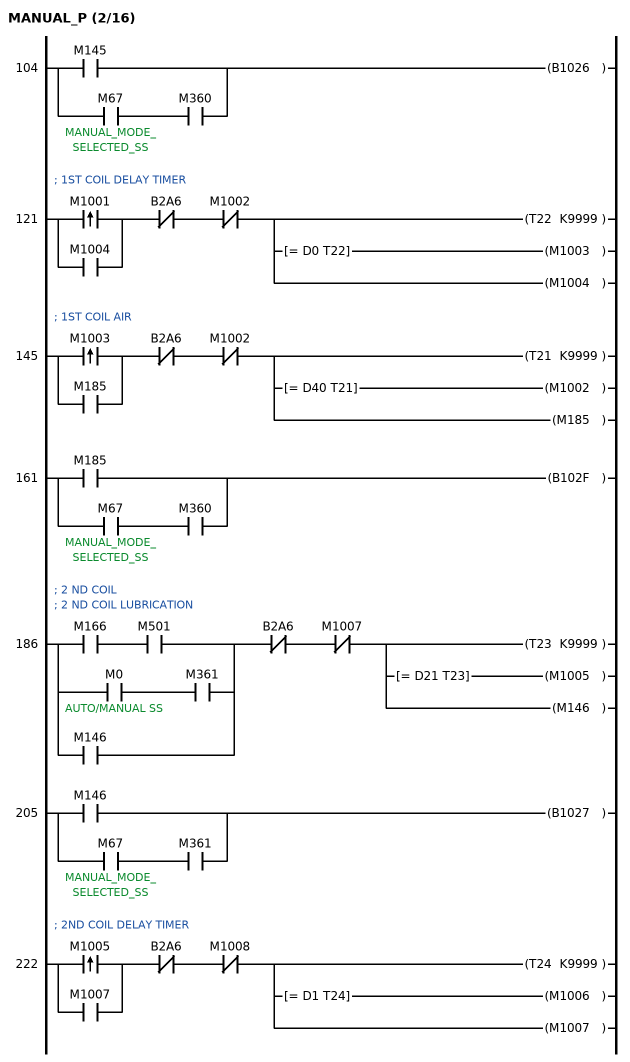
[picture p24: ladder of MANUAL_P, rungs at steps 104 to 222]
104   LD      M145
      LD      M67  ; MANUAL_MODE_SELECTED_SS
      AND     M360
      ORB
      OUT     B1026
; 1ST COIL DELAY TIMER
121   LDP     M1001
      OR      M1004
      ANI     B2A6
      ANI     M1002
      OUT     T22 K9999
      MPS
      AND=    D0 T22
      OUT     M1003
      MPP
      OUT     M1004
; 1ST COIL AIR
145   LDP     M1003
      OR      M185
      ANI     B2A6
      ANI     M1002
      OUT     T21 K9999
      MPS
      AND=    D40 T21
      OUT     M1002
      MPP
      OUT     M185
161   LD      M185
      LD      M67  ; MANUAL_MODE_SELECTED_SS
      AND     M360
      ORB
      OUT     B102F
; 2 ND COIL
; 2 ND COIL LUBRICATION
186   LD      M166
      AND     M501
      LD      M0  ; AUTO/MANUAL SS
      AND     M361
      ORB
      OR      M146
      ANI     B2A6
      ANI     M1007
      OUT     T23 K9999
      MPS
      AND=    D21 T23
      OUT     M1005
      MPP
      OUT     M146
205   LD      M146
      LD      M67  ; MANUAL_MODE_SELECTED_SS
      AND     M361
      ORB
      OUT     B1027
; 2ND COIL DELAY TIMER
222   LDP     M1005
      OR      M1007
      ANI     B2A6
      ANI     M1008
      OUT     T24 K9999
      MPS
      AND=    D1 T24
      OUT     M1006
      MPP
      OUT     M1007
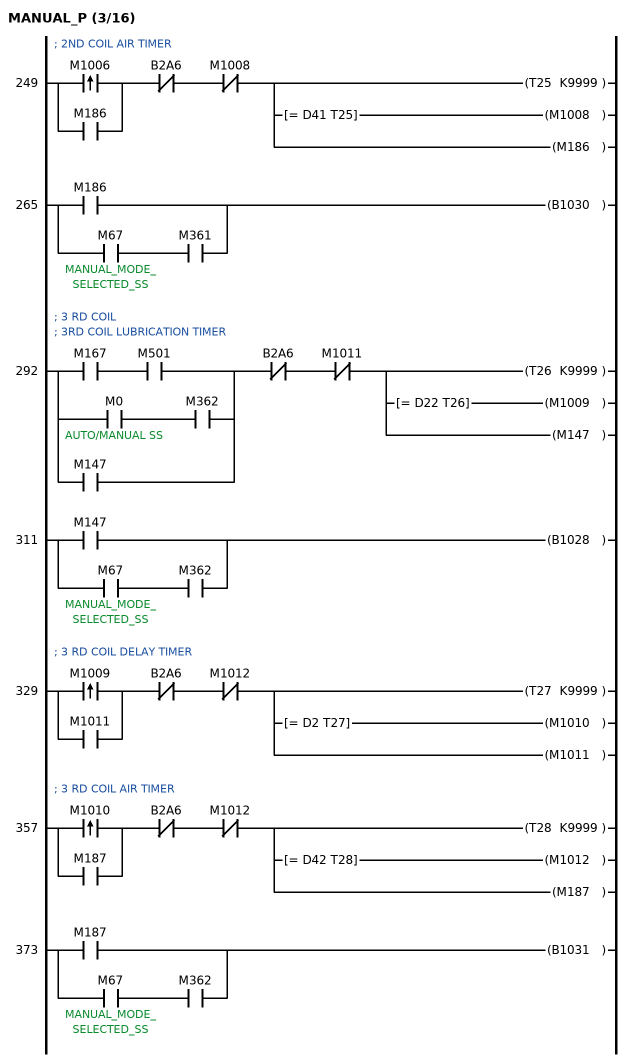
; 2ND COIL AIR TIMER
249   LDP     M1006
      OR      M186
      ANI     B2A6
      ANI     M1008
      OUT     T25 K9999
      MPS
      AND=    D41 T25
      OUT     M1008
      MPP
      OUT     M186
265   LD      M186
      LD      M67  ; MANUAL_MODE_SELECTED_SS
      AND     M361
      ORB
      OUT     B1030
; 3 RD COIL
; 3RD COIL LUBRICATION TIMER
292   LD      M167
      AND     M501
      LD      M0  ; AUTO/MANUAL SS
      AND     M362
      ORB
      OR      M147
      ANI     B2A6
      ANI     M1011
      OUT     T26 K9999
      MPS
      AND=    D22 T26
      OUT     M1009
      MPP
      OUT     M147
311   LD      M147
      LD      M67  ; MANUAL_MODE_SELECTED_SS
      AND     M362
      ORB
      OUT     B1028
; 3 RD COIL DELAY TIMER
329   LDP     M1009
      OR      M1011
      ANI     B2A6
      ANI     M1012
      OUT     T27 K9999
      MPS
      AND=    D2 T27
      OUT     M1010
      MPP
      OUT     M1011
; 3 RD COIL AIR TIMER
357   LDP     M1010
      OR      M187
      ANI     B2A6
      ANI     M1012
      OUT     T28 K9999
      MPS
      AND=    D42 T28
      OUT     M1012
      MPP
      OUT     M187
373   LD      M187
      LD      M67  ; MANUAL_MODE_SELECTED_SS
      AND     M362
      ORB
      OUT     B1031
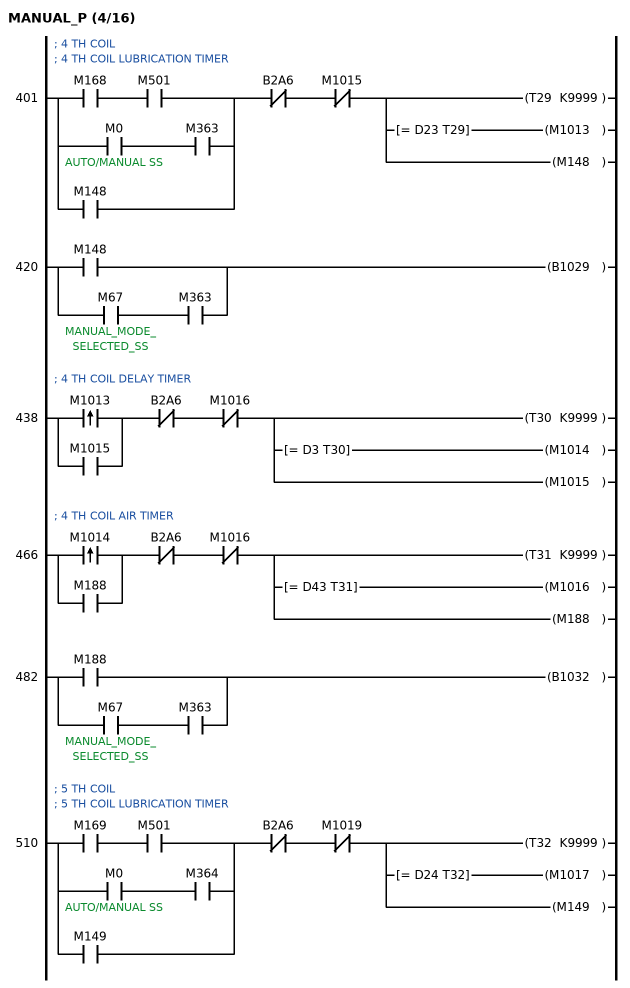
; 4 TH COIL
; 4 TH COIL LUBRICATION TIMER
401   LD      M168
      AND     M501
      LD      M0  ; AUTO/MANUAL SS
      AND     M363
      ORB
      OR      M148
      ANI     B2A6
      ANI     M1015
      OUT     T29 K9999
      MPS
      AND=    D23 T29
      OUT     M1013
      MPP
      OUT     M148
420   LD      M148
      LD      M67  ; MANUAL_MODE_SELECTED_SS
      AND     M363
      ORB
      OUT     B1029
; 4 TH COIL DELAY TIMER
438   LDP     M1013
      OR      M1015
      ANI     B2A6
      ANI     M1016
      OUT     T30 K9999
      MPS
      AND=    D3 T30
      OUT     M1014
      MPP
      OUT     M1015
; 4 TH COIL AIR TIMER
466   LDP     M1014
      OR      M188
      ANI     B2A6
      ANI     M1016
      OUT     T31 K9999
      MPS
      AND=    D43 T31
      OUT     M1016
      MPP
      OUT     M188
482   LD      M188
      LD      M67  ; MANUAL_MODE_SELECTED_SS
      AND     M363
      ORB
      OUT     B1032
; 5 TH COIL
; 5 TH COIL LUBRICATION TIMER
510   LD      M169
      AND     M501
      LD      M0  ; AUTO/MANUAL SS
      AND     M364
      ORB
      OR      M149
      ANI     B2A6
      ANI     M1019
      OUT     T32 K9999
      MPS
      AND=    D24 T32
      OUT     M1017
      MPP
      OUT     M149
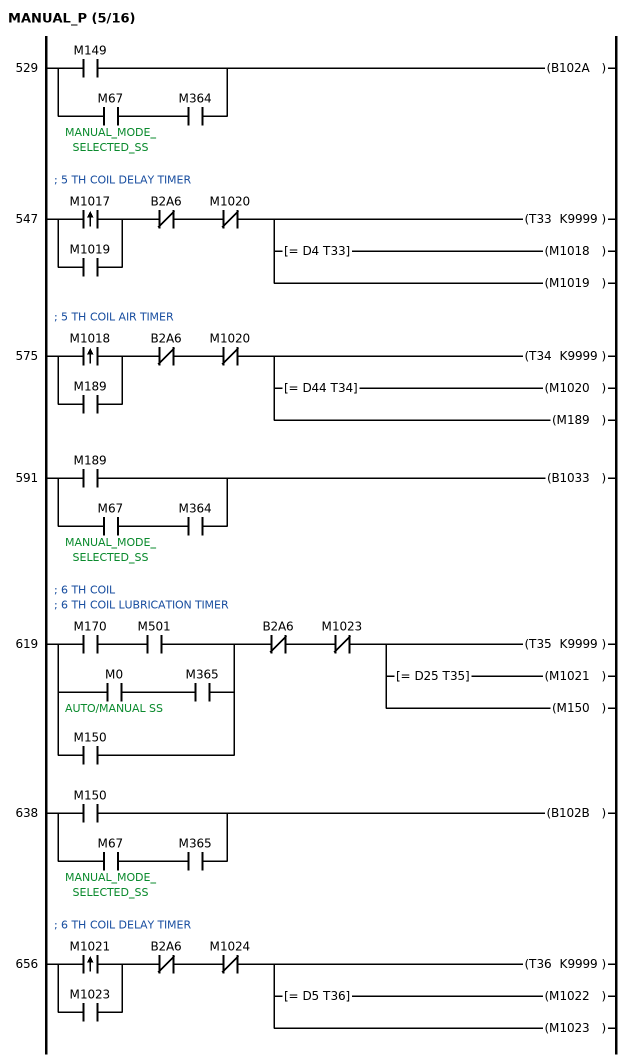
529   LD      M149
      LD      M67  ; MANUAL_MODE_SELECTED_SS
      AND     M364
      ORB
      OUT     B102A
; 5 TH COIL DELAY TIMER
547   LDP     M1017
      OR      M1019
      ANI     B2A6
      ANI     M1020
      OUT     T33 K9999
      MPS
      AND=    D4 T33
      OUT     M1018
      MPP
      OUT     M1019
; 5 TH COIL AIR TIMER
575   LDP     M1018
      OR      M189
      ANI     B2A6
      ANI     M1020
      OUT     T34 K9999
      MPS
      AND=    D44 T34
      OUT     M1020
      MPP
      OUT     M189
591   LD      M189
      LD      M67  ; MANUAL_MODE_SELECTED_SS
      AND     M364
      ORB
      OUT     B1033
; 6 TH COIL
; 6 TH COIL LUBRICATION TIMER
619   LD      M170
      AND     M501
      LD      M0  ; AUTO/MANUAL SS
      AND     M365
      ORB
      OR      M150
      ANI     B2A6
      ANI     M1023
      OUT     T35 K9999
      MPS
      AND=    D25 T35
      OUT     M1021
      MPP
      OUT     M150
638   LD      M150
      LD      M67  ; MANUAL_MODE_SELECTED_SS
      AND     M365
      ORB
      OUT     B102B
; 6 TH COIL DELAY TIMER
656   LDP     M1021
      OR      M1023
      ANI     B2A6
      ANI     M1024
      OUT     T36 K9999
      MPS
      AND=    D5 T36
      OUT     M1022
      MPP
      OUT     M1023
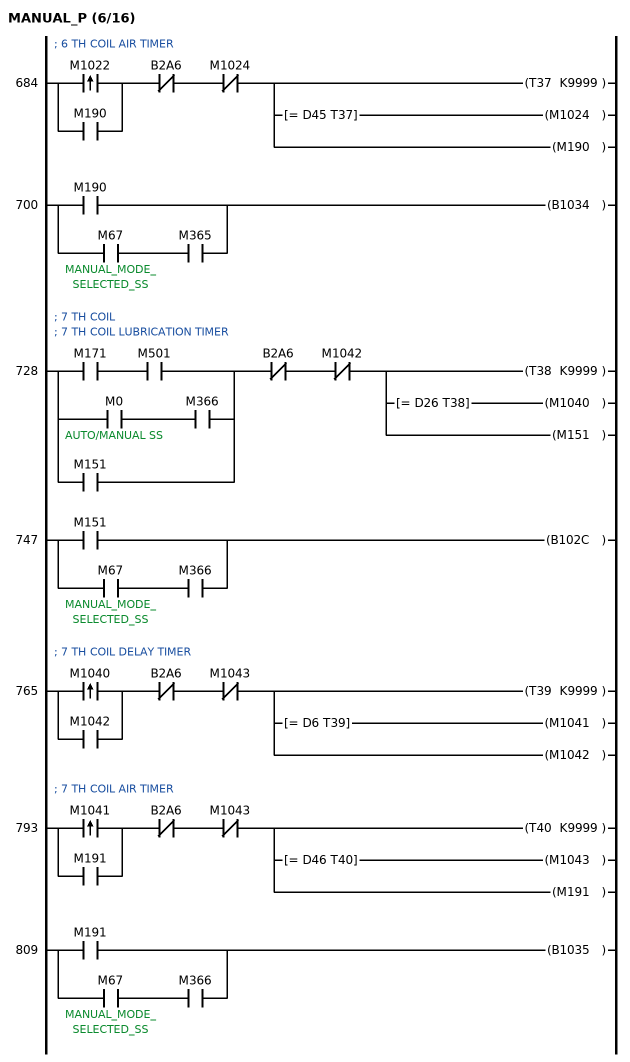
; 6 TH COIL AIR TIMER
684   LDP     M1022
      OR      M190
      ANI     B2A6
      ANI     M1024
      OUT     T37 K9999
      MPS
      AND=    D45 T37
      OUT     M1024
      MPP
      OUT     M190
700   LD      M190
      LD      M67  ; MANUAL_MODE_SELECTED_SS
      AND     M365
      ORB
      OUT     B1034
; 7 TH COIL
; 7 TH COIL LUBRICATION TIMER
728   LD      M171
      AND     M501
      LD      M0  ; AUTO/MANUAL SS
      AND     M366
      ORB
      OR      M151
      ANI     B2A6
      ANI     M1042
      OUT     T38 K9999
      MPS
      AND=    D26 T38
      OUT     M1040
      MPP
      OUT     M151
747   LD      M151
      LD      M67  ; MANUAL_MODE_SELECTED_SS
      AND     M366
      ORB
      OUT     B102C
; 7 TH COIL DELAY TIMER
765   LDP     M1040
      OR      M1042
      ANI     B2A6
      ANI     M1043
      OUT     T39 K9999
      MPS
      AND=    D6 T39
      OUT     M1041
      MPP
      OUT     M1042
; 7 TH COIL AIR TIMER
793   LDP     M1041
      OR      M191
      ANI     B2A6
      ANI     M1043
      OUT     T40 K9999
      MPS
      AND=    D46 T40
      OUT     M1043
      MPP
      OUT     M191
809   LD      M191
      LD      M67  ; MANUAL_MODE_SELECTED_SS
      AND     M366
      ORB
      OUT     B1035
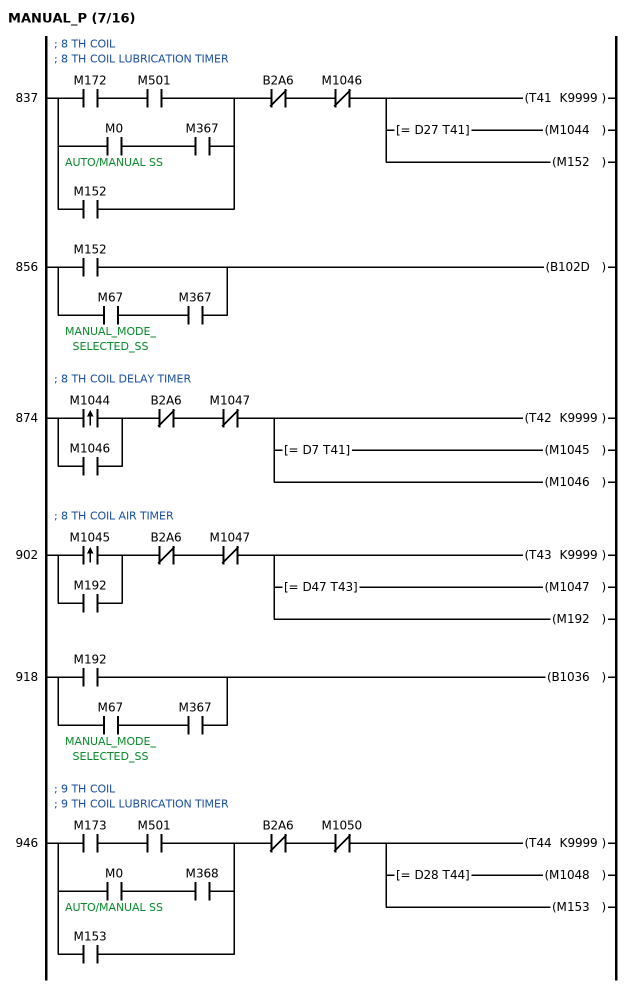
; 8 TH COIL
; 8 TH COIL LUBRICATION TIMER
837   LD      M172
      AND     M501
      LD      M0  ; AUTO/MANUAL SS
      AND     M367
      ORB
      OR      M152
      ANI     B2A6
      ANI     M1046
      OUT     T41 K9999
      MPS
      AND=    D27 T41
      OUT     M1044
      MPP
      OUT     M152
856   LD      M152
      LD      M67  ; MANUAL_MODE_SELECTED_SS
      AND     M367
      ORB
      OUT     B102D
; 8 TH COIL DELAY TIMER
874   LDP     M1044
      OR      M1046
      ANI     B2A6
      ANI     M1047
      OUT     T42 K9999
      MPS
      AND=    D7 T41
      OUT     M1045
      MPP
      OUT     M1046
; 8 TH COIL AIR TIMER
902   LDP     M1045
      OR      M192
      ANI     B2A6
      ANI     M1047
      OUT     T43 K9999
      MPS
      AND=    D47 T43
      OUT     M1047
      MPP
      OUT     M192
918   LD      M192
      LD      M67  ; MANUAL_MODE_SELECTED_SS
      AND     M367
      ORB
      OUT     B1036
; 9 TH COIL
; 9 TH COIL LUBRICATION TIMER
946   LD      M173
      AND     M501
      LD      M0  ; AUTO/MANUAL SS
      AND     M368
      ORB
      OR      M153
      ANI     B2A6
      ANI     M1050
      OUT     T44 K9999
      MPS
      AND=    D28 T44
      OUT     M1048
      MPP
      OUT     M153
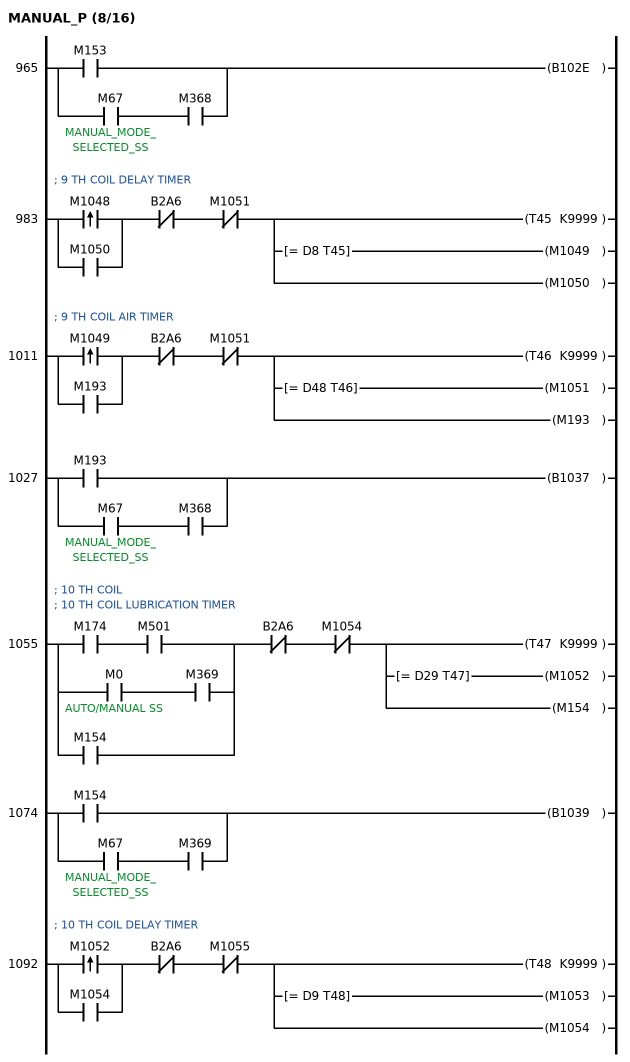
965   LD      M153
      LD      M67  ; MANUAL_MODE_SELECTED_SS
      AND     M368
      ORB
      OUT     B102E
; 9 TH COIL DELAY TIMER
983   LDP     M1048
      OR      M1050
      ANI     B2A6
      ANI     M1051
      OUT     T45 K9999
      MPS
      AND=    D8 T45
      OUT     M1049
      MPP
      OUT     M1050
; 9 TH COIL AIR TIMER
1011  LDP     M1049
      OR      M193
      ANI     B2A6
      ANI     M1051
      OUT     T46 K9999
      MPS
      AND=    D48 T46
      OUT     M1051
      MPP
      OUT     M193
1027  LD      M193
      LD      M67  ; MANUAL_MODE_SELECTED_SS
      AND     M368
      ORB
      OUT     B1037
; 10 TH COIL
; 10 TH COIL LUBRICATION TIMER
1055  LD      M174
      AND     M501
      LD      M0  ; AUTO/MANUAL SS
      AND     M369
      ORB
      OR      M154
      ANI     B2A6
      ANI     M1054
      OUT     T47 K9999
      MPS
      AND=    D29 T47
      OUT     M1052
      MPP
      OUT     M154
1074  LD      M154
      LD      M67  ; MANUAL_MODE_SELECTED_SS
      AND     M369
      ORB
      OUT     B1039
; 10 TH COIL DELAY TIMER
1092  LDP     M1052
      OR      M1054
      ANI     B2A6
      ANI     M1055
      OUT     T48 K9999
      MPS
      AND=    D9 T48
      OUT     M1053
      MPP
      OUT     M1054
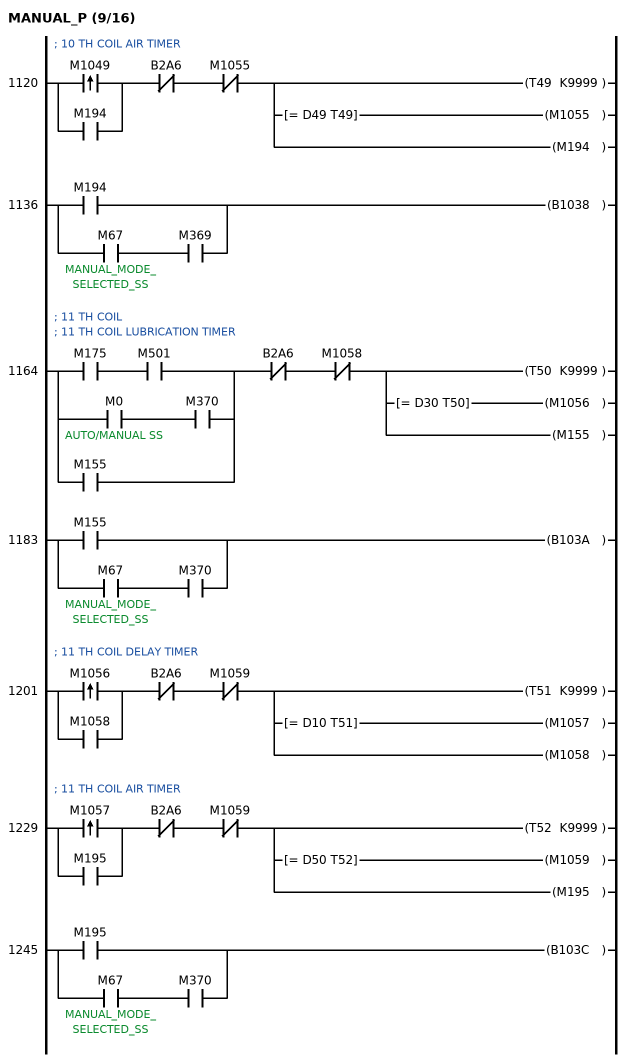
; 10 TH COIL AIR TIMER
1120  LDP     M1049
      OR      M194
      ANI     B2A6
      ANI     M1055
      OUT     T49 K9999
      MPS
      AND=    D49 T49
      OUT     M1055
      MPP
      OUT     M194
1136  LD      M194
      LD      M67  ; MANUAL_MODE_SELECTED_SS
      AND     M369
      ORB
      OUT     B1038
; 11 TH COIL
; 11 TH COIL LUBRICATION TIMER
1164  LD      M175
      AND     M501
      LD      M0  ; AUTO/MANUAL SS
      AND     M370
      ORB
      OR      M155
      ANI     B2A6
      ANI     M1058
      OUT     T50 K9999
      MPS
      AND=    D30 T50
      OUT     M1056
      MPP
      OUT     M155
1183  LD      M155
      LD      M67  ; MANUAL_MODE_SELECTED_SS
      AND     M370
      ORB
      OUT     B103A
; 11 TH COIL DELAY TIMER
1201  LDP     M1056
      OR      M1058
      ANI     B2A6
      ANI     M1059
      OUT     T51 K9999
      MPS
      AND=    D10 T51
      OUT     M1057
      MPP
      OUT     M1058
; 11 TH COIL AIR TIMER
1229  LDP     M1057
      OR      M195
      ANI     B2A6
      ANI     M1059
      OUT     T52 K9999
      MPS
      AND=    D50 T52
      OUT     M1059
      MPP
      OUT     M195
1245  LD      M195
      LD      M67  ; MANUAL_MODE_SELECTED_SS
      AND     M370
      ORB
      OUT     B103C
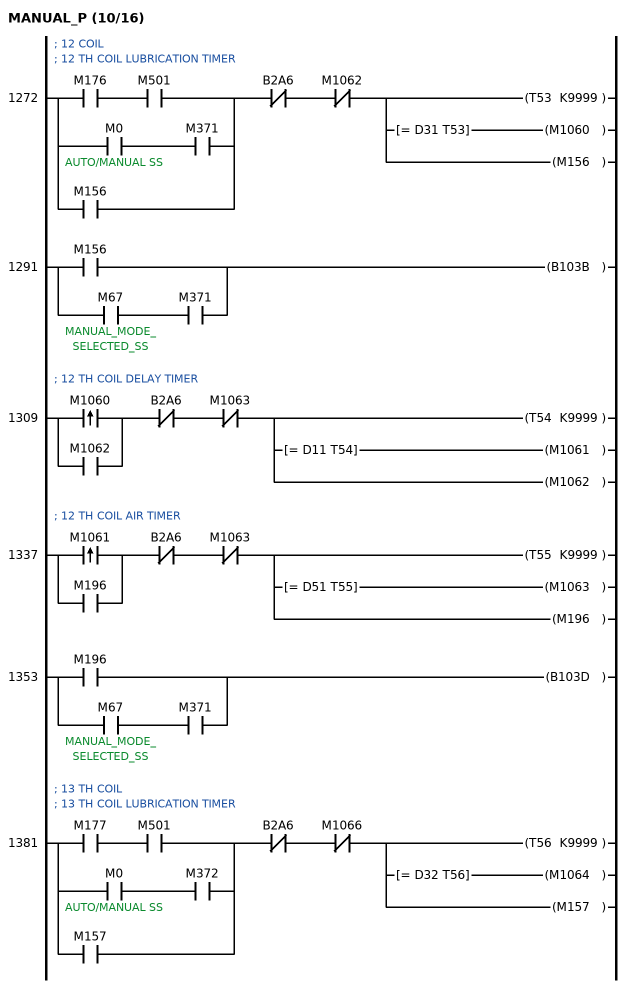
; 12 COIL
; 12 TH COIL LUBRICATION TIMER
1272  LD      M176
      AND     M501
      LD      M0  ; AUTO/MANUAL SS
      AND     M371
      ORB
      OR      M156
      ANI     B2A6
      ANI     M1062
      OUT     T53 K9999
      MPS
      AND=    D31 T53
      OUT     M1060
      MPP
      OUT     M156
1291  LD      M156
      LD      M67  ; MANUAL_MODE_SELECTED_SS
      AND     M371
      ORB
      OUT     B103B
; 12 TH COIL DELAY TIMER
1309  LDP     M1060
      OR      M1062
      ANI     B2A6
      ANI     M1063
      OUT     T54 K9999
      MPS
      AND=    D11 T54
      OUT     M1061
      MPP
      OUT     M1062
; 12 TH COIL AIR TIMER
1337  LDP     M1061
      OR      M196
      ANI     B2A6
      ANI     M1063
      OUT     T55 K9999
      MPS
      AND=    D51 T55
      OUT     M1063
      MPP
      OUT     M196
1353  LD      M196
      LD      M67  ; MANUAL_MODE_SELECTED_SS
      AND     M371
      ORB
      OUT     B103D
; 13 TH COIL
; 13 TH COIL LUBRICATION TIMER
1381  LD      M177
      AND     M501
      LD      M0  ; AUTO/MANUAL SS
      AND     M372
      ORB
      OR      M157
      ANI     B2A6
      ANI     M1066
      OUT     T56 K9999
      MPS
      AND=    D32 T56
      OUT     M1064
      MPP
      OUT     M157
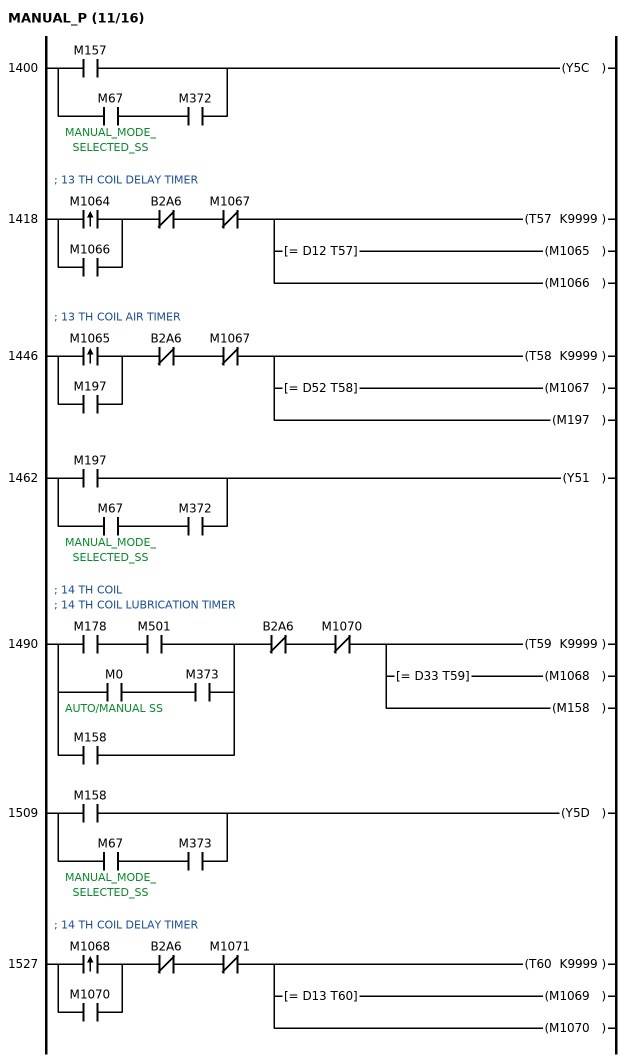
1400  LD      M157
      LD      M67  ; MANUAL_MODE_SELECTED_SS
      AND     M372
      ORB
      OUT     Y5C
; 13 TH COIL DELAY TIMER
1418  LDP     M1064
      OR      M1066
      ANI     B2A6
      ANI     M1067
      OUT     T57 K9999
      MPS
      AND=    D12 T57
      OUT     M1065
      MPP
      OUT     M1066
; 13 TH COIL AIR TIMER
1446  LDP     M1065
      OR      M197
      ANI     B2A6
      ANI     M1067
      OUT     T58 K9999
      MPS
      AND=    D52 T58
      OUT     M1067
      MPP
      OUT     M197
1462  LD      M197
      LD      M67  ; MANUAL_MODE_SELECTED_SS
      AND     M372
      ORB
      OUT     Y51
; 14 TH COIL
; 14 TH COIL LUBRICATION TIMER
1490  LD      M178
      AND     M501
      LD      M0  ; AUTO/MANUAL SS
      AND     M373
      ORB
      OR      M158
      ANI     B2A6
      ANI     M1070
      OUT     T59 K9999
      MPS
      AND=    D33 T59
      OUT     M1068
      MPP
      OUT     M158
1509  LD      M158
      LD      M67  ; MANUAL_MODE_SELECTED_SS
      AND     M373
      ORB
      OUT     Y5D
; 14 TH COIL DELAY TIMER
1527  LDP     M1068
      OR      M1070
      ANI     B2A6
      ANI     M1071
      OUT     T60 K9999
      MPS
      AND=    D13 T60
      OUT     M1069
      MPP
      OUT     M1070
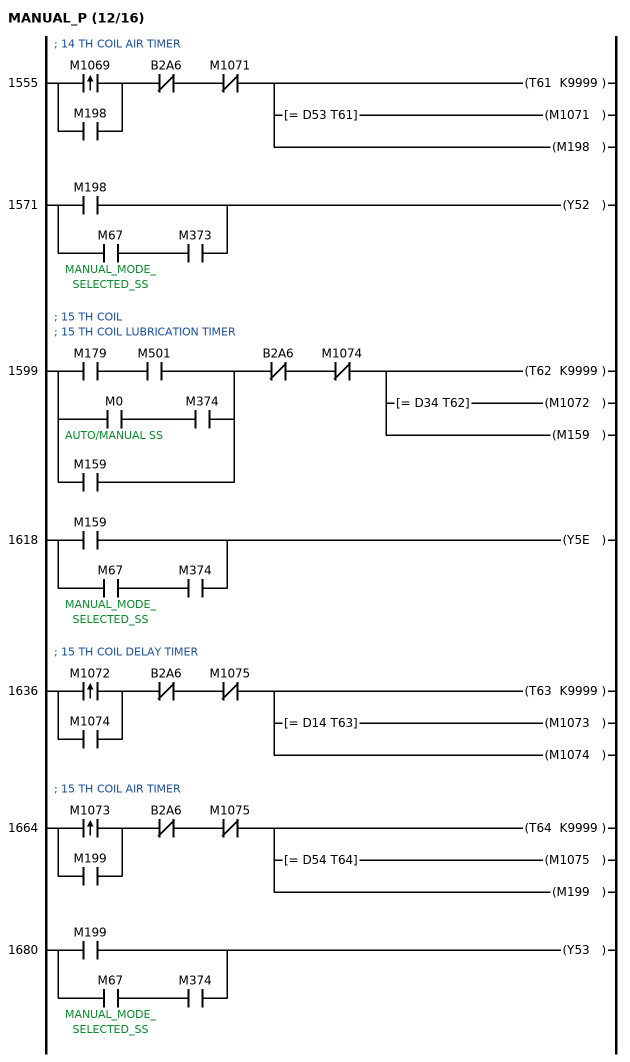
; 14 TH COIL AIR TIMER
1555  LDP     M1069
      OR      M198
      ANI     B2A6
      ANI     M1071
      OUT     T61 K9999
      MPS
      AND=    D53 T61
      OUT     M1071
      MPP
      OUT     M198
1571  LD      M198
      LD      M67  ; MANUAL_MODE_SELECTED_SS
      AND     M373
      ORB
      OUT     Y52
; 15 TH COIL
; 15 TH COIL LUBRICATION TIMER
1599  LD      M179
      AND     M501
      LD      M0  ; AUTO/MANUAL SS
      AND     M374
      ORB
      OR      M159
      ANI     B2A6
      ANI     M1074
      OUT     T62 K9999
      MPS
      AND=    D34 T62
      OUT     M1072
      MPP
      OUT     M159
1618  LD      M159
      LD      M67  ; MANUAL_MODE_SELECTED_SS
      AND     M374
      ORB
      OUT     Y5E
; 15 TH COIL DELAY TIMER
1636  LDP     M1072
      OR      M1074
      ANI     B2A6
      ANI     M1075
      OUT     T63 K9999
      MPS
      AND=    D14 T63
      OUT     M1073
      MPP
      OUT     M1074
; 15 TH COIL AIR TIMER
1664  LDP     M1073
      OR      M199
      ANI     B2A6
      ANI     M1075
      OUT     T64 K9999
      MPS
      AND=    D54 T64
      OUT     M1075
      MPP
      OUT     M199
1680  LD      M199
      LD      M67  ; MANUAL_MODE_SELECTED_SS
      AND     M374
      ORB
      OUT     Y53
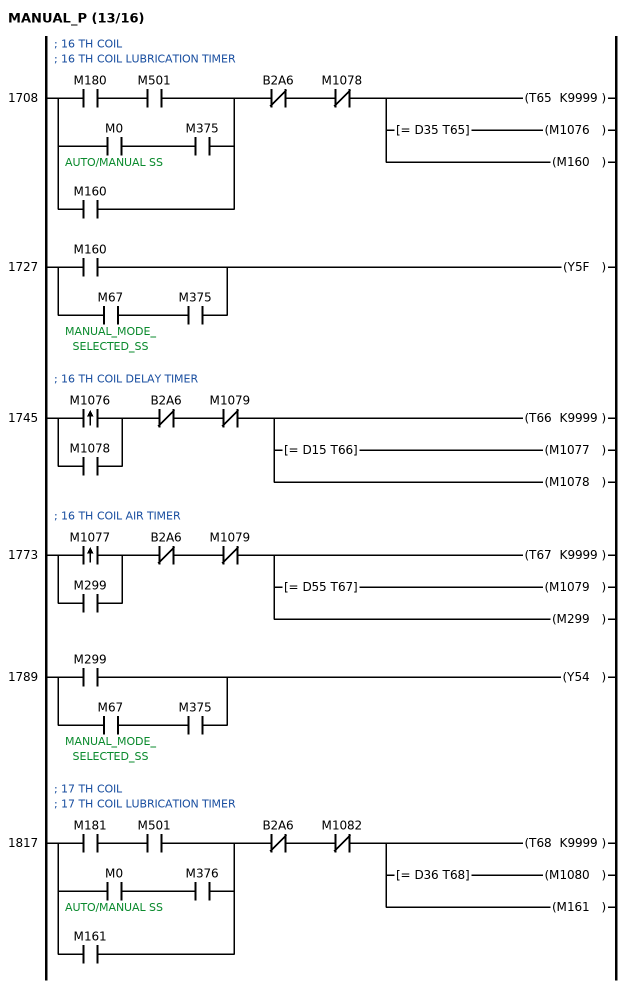
; 16 TH COIL
; 16 TH COIL LUBRICATION TIMER
1708  LD      M180
      AND     M501
      LD      M0  ; AUTO/MANUAL SS
      AND     M375
      ORB
      OR      M160
      ANI     B2A6
      ANI     M1078
      OUT     T65 K9999
      MPS
      AND=    D35 T65
      OUT     M1076
      MPP
      OUT     M160
1727  LD      M160
      LD      M67  ; MANUAL_MODE_SELECTED_SS
      AND     M375
      ORB
      OUT     Y5F
; 16 TH COIL DELAY TIMER
1745  LDP     M1076
      OR      M1078
      ANI     B2A6
      ANI     M1079
      OUT     T66 K9999
      MPS
      AND=    D15 T66
      OUT     M1077
      MPP
      OUT     M1078
; 16 TH COIL AIR TIMER
1773  LDP     M1077
      OR      M299
      ANI     B2A6
      ANI     M1079
      OUT     T67 K9999
      MPS
      AND=    D55 T67
      OUT     M1079
      MPP
      OUT     M299
1789  LD      M299
      LD      M67  ; MANUAL_MODE_SELECTED_SS
      AND     M375
      ORB
      OUT     Y54
; 17 TH COIL
; 17 TH COIL LUBRICATION TIMER
1817  LD      M181
      AND     M501
      LD      M0  ; AUTO/MANUAL SS
      AND     M376
      ORB
      OR      M161
      ANI     B2A6
      ANI     M1082
      OUT     T68 K9999
      MPS
      AND=    D36 T68
      OUT     M1080
      MPP
      OUT     M161
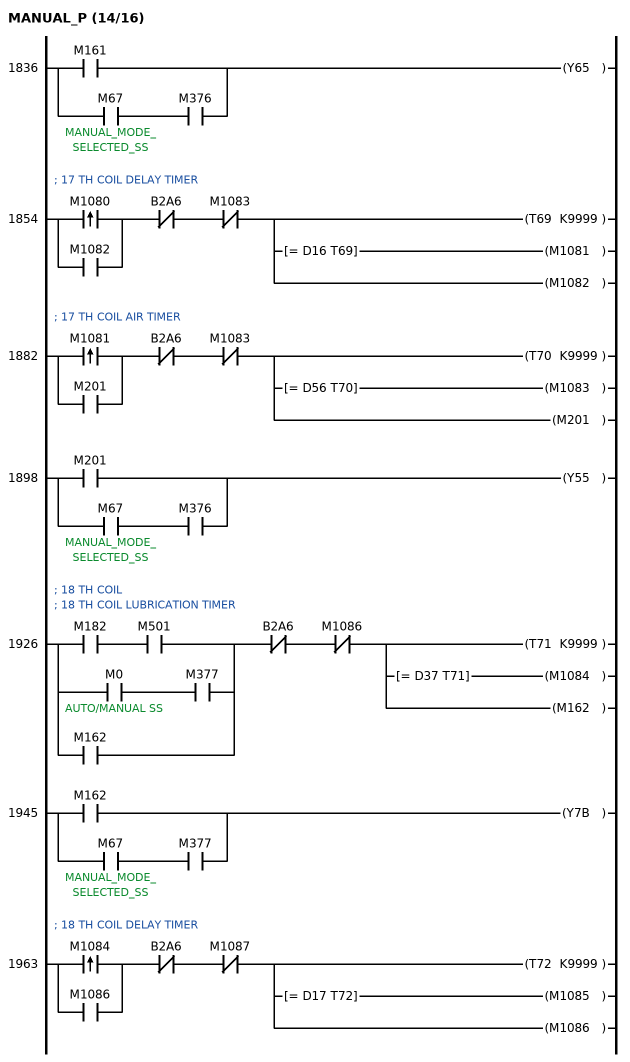
1836  LD      M161
      LD      M67  ; MANUAL_MODE_SELECTED_SS
      AND     M376
      ORB
      OUT     Y65
; 17 TH COIL DELAY TIMER
1854  LDP     M1080
      OR      M1082
      ANI     B2A6
      ANI     M1083
      OUT     T69 K9999
      MPS
      AND=    D16 T69
      OUT     M1081
      MPP
      OUT     M1082
; 17 TH COIL AIR TIMER
1882  LDP     M1081
      OR      M201
      ANI     B2A6
      ANI     M1083
      OUT     T70 K9999
      MPS
      AND=    D56 T70
      OUT     M1083
      MPP
      OUT     M201
1898  LD      M201
      LD      M67  ; MANUAL_MODE_SELECTED_SS
      AND     M376
      ORB
      OUT     Y55
; 18 TH COIL
; 18 TH COIL LUBRICATION TIMER
1926  LD      M182
      AND     M501
      LD      M0  ; AUTO/MANUAL SS
      AND     M377
      ORB
      OR      M162
      ANI     B2A6
      ANI     M1086
      OUT     T71 K9999
      MPS
      AND=    D37 T71
      OUT     M1084
      MPP
      OUT     M162
1945  LD      M162
      LD      M67  ; MANUAL_MODE_SELECTED_SS
      AND     M377
      ORB
      OUT     Y7B
; 18 TH COIL DELAY TIMER
1963  LDP     M1084
      OR      M1086
      ANI     B2A6
      ANI     M1087
      OUT     T72 K9999
      MPS
      AND=    D17 T72
      OUT     M1085
      MPP
      OUT     M1086
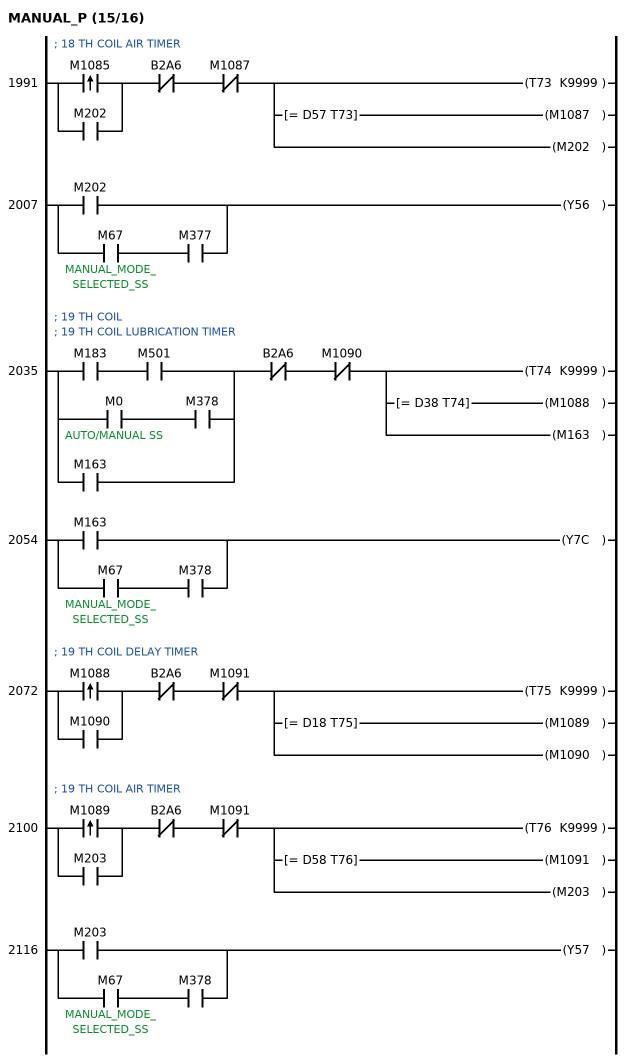
; 18 TH COIL AIR TIMER
1991  LDP     M1085
      OR      M202
      ANI     B2A6
      ANI     M1087
      OUT     T73 K9999
      MPS
      AND=    D57 T73
      OUT     M1087
      MPP
      OUT     M202
2007  LD      M202
      LD      M67  ; MANUAL_MODE_SELECTED_SS
      AND     M377
      ORB
      OUT     Y56
; 19 TH COIL
; 19 TH COIL LUBRICATION TIMER
2035  LD      M183
      AND     M501
      LD      M0  ; AUTO/MANUAL SS
      AND     M378
      ORB
      OR      M163
      ANI     B2A6
      ANI     M1090
      OUT     T74 K9999
      MPS
      AND=    D38 T74
      OUT     M1088
      MPP
      OUT     M163
2054  LD      M163
      LD      M67  ; MANUAL_MODE_SELECTED_SS
      AND     M378
      ORB
      OUT     Y7C
; 19 TH COIL DELAY TIMER
2072  LDP     M1088
      OR      M1090
      ANI     B2A6
      ANI     M1091
      OUT     T75 K9999
      MPS
      AND=    D18 T75
      OUT     M1089
      MPP
      OUT     M1090
; 19 TH COIL AIR TIMER
2100  LDP     M1089
      OR      M203
      ANI     B2A6
      ANI     M1091
      OUT     T76 K9999
      MPS
      AND=    D58 T76
      OUT     M1091
      MPP
      OUT     M203
2116  LD      M203
      LD      M67  ; MANUAL_MODE_SELECTED_SS
      AND     M378
      ORB
      OUT     Y57
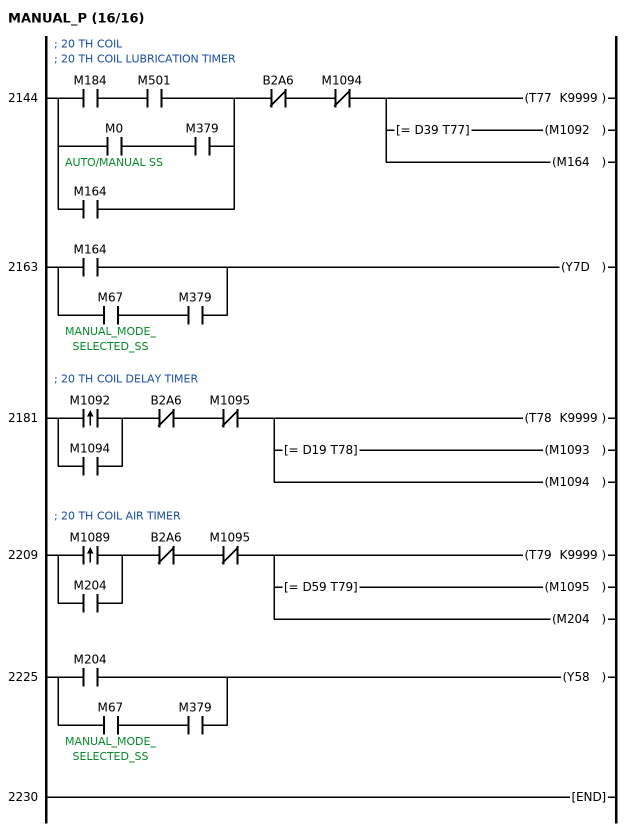
; 20 TH COIL
; 20 TH COIL LUBRICATION TIMER
2144  LD      M184
      AND     M501
      LD      M0  ; AUTO/MANUAL SS
      AND     M379
      ORB
      OR      M164
      ANI     B2A6
      ANI     M1094
      OUT     T77 K9999
      MPS
      AND=    D39 T77
      OUT     M1092
      MPP
      OUT     M164
2163  LD      M164
      LD      M67  ; MANUAL_MODE_SELECTED_SS
      AND     M379
      ORB
      OUT     Y7D
; 20 TH COIL DELAY TIMER
2181  LDP     M1092
      OR      M1094
      ANI     B2A6
      ANI     M1095
      OUT     T78 K9999
      MPS
      AND=    D19 T78
      OUT     M1093
      MPP
      OUT     M1094
; 20 TH COIL AIR TIMER
2209  LDP     M1089
      OR      M204
      ANI     B2A6
      ANI     M1095
      OUT     T79 K9999
      MPS
      AND=    D59 T79
      OUT     M1095
      MPP
      OUT     M204
2225  LD      M204
      LD      M67  ; MANUAL_MODE_SELECTED_SS
      AND     M379
      ORB
      OUT     Y58
2230  END
END_PROGRAM

PROGRAM OUTPUT_M
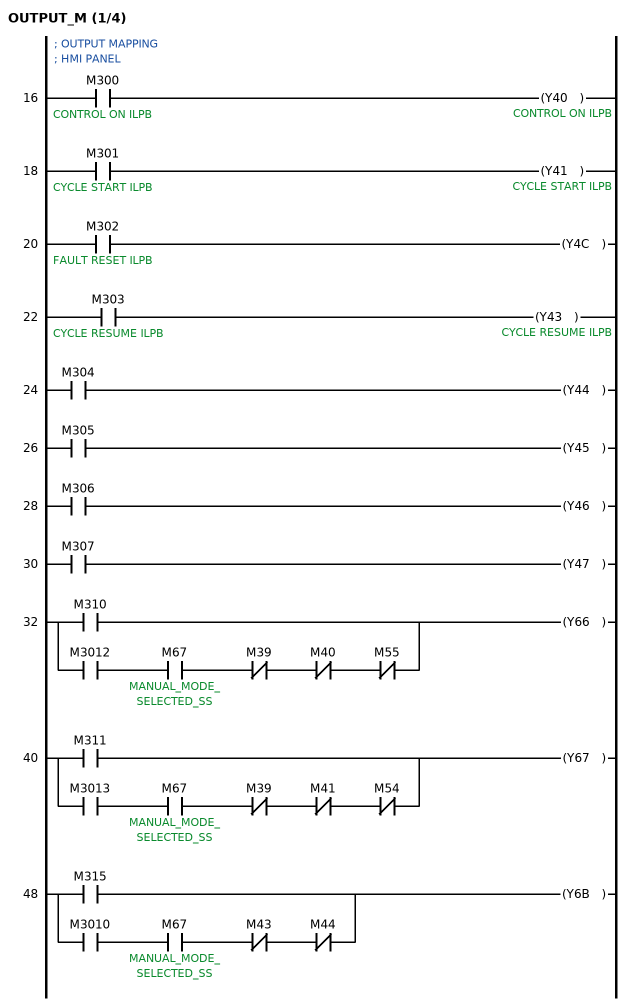
; OUTPUT MAPPING
; HMI PANEL
16    LD      M300  ; CONTROL ON ILPB
      OUT     Y40  ; CONTROL ON ILPB
18    LD      M301  ; CYCLE START ILPB
      OUT     Y41  ; CYCLE START ILPB
20    LD      M302  ; FAULT RESET ILPB
      OUT     Y4C
22    LD      M303  ; CYCLE RESUME ILPB
      OUT     Y43  ; CYCLE RESUME ILPB
24    LD      M304
      OUT     Y44
26    LD      M305
      OUT     Y45
28    LD      M306
      OUT     Y46
30    LD      M307
      OUT     Y47
32    LD      M310
      LD      M3012
      AND     M67  ; MANUAL_MODE_SELECTED_SS
      ANI     M39
      ANI     M40
      ANI     M55
      ORB
      OUT     Y66
40    LD      M311
      LD      M3013
      AND     M67  ; MANUAL_MODE_SELECTED_SS
      ANI     M39
      ANI     M41
      ANI     M54
      ORB
      OUT     Y67
48    LD      M315
      LD      M3010
      AND     M67  ; MANUAL_MODE_SELECTED_SS
      ANI     M43
      ANI     M44
      ORB
      OUT     Y6B
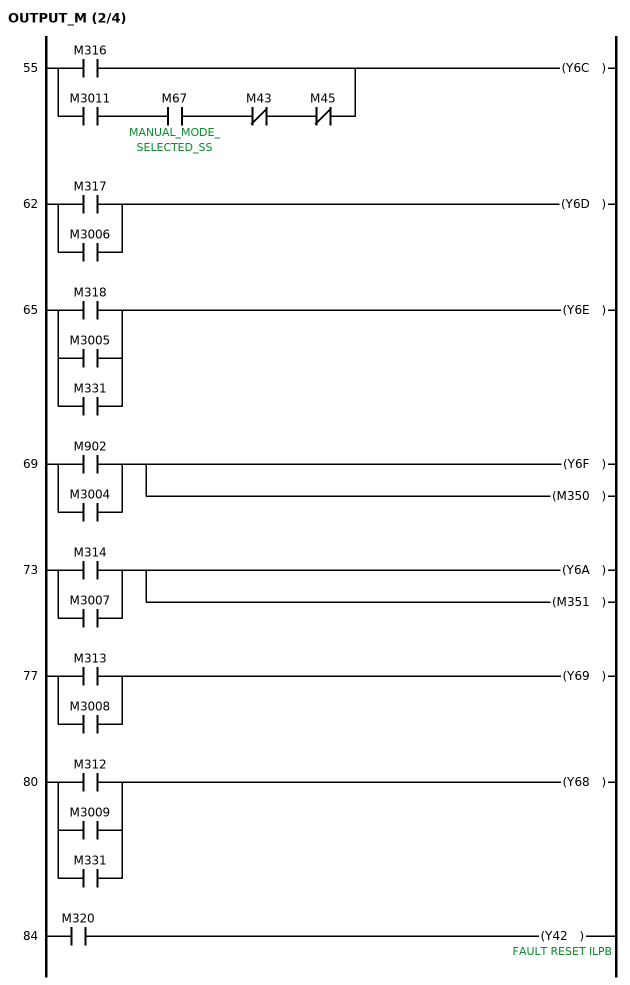
55    LD      M316
      LD      M3011
      AND     M67  ; MANUAL_MODE_SELECTED_SS
      ANI     M43
      ANI     M45
      ORB
      OUT     Y6C
62    LD      M317
      OR      M3006
      OUT     Y6D
65    LD      M318
      OR      M3005
      OR      M331
      OUT     Y6E
69    LD      M902
      OR      M3004
      OUT     Y6F
      OUT     M350
73    LD      M314
      OR      M3007
      OUT     Y6A
      OUT     M351
77    LD      M313
      OR      M3008
      OUT     Y69
80    LD      M312
      OR      M3009
      OR      M331
      OUT     Y68
84    LD      M320
      OUT     Y42  ; FAULT RESET ILPB
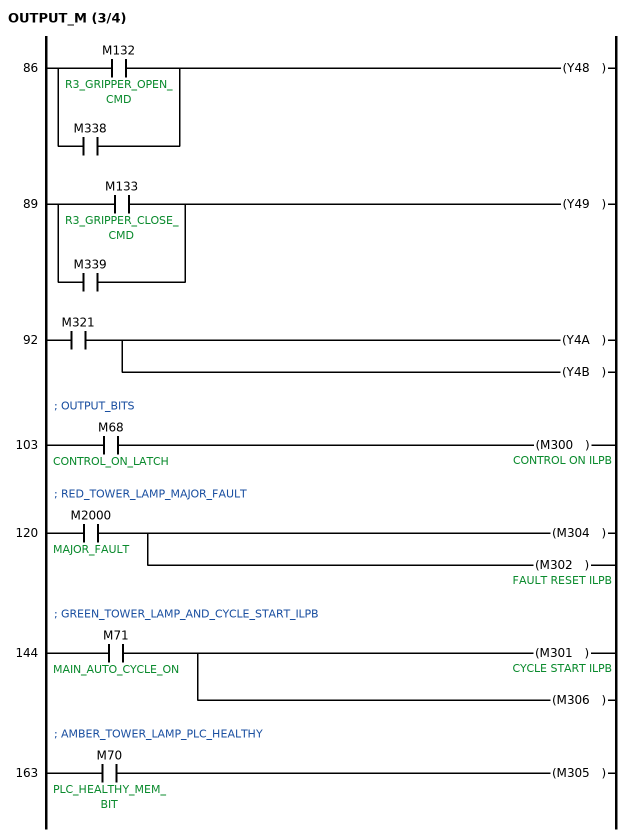
86    LD      M132  ; R3_GRIPPER_OPEN_CMD
      OR      M338
      OUT     Y48
89    LD      M133  ; R3_GRIPPER_CLOSE_CMD
      OR      M339
      OUT     Y49
92    LD      M321
      OUT     Y4A
      OUT     Y4B
; OUTPUT_BITS
103   LD      M68  ; CONTROL_ON_LATCH
      OUT     M300  ; CONTROL ON ILPB
; RED_TOWER_LAMP_MAJOR_FAULT
120   LD      M2000  ; MAJOR_FAULT
      OUT     M304
      OUT     M302  ; FAULT RESET ILPB
; GREEN_TOWER_LAMP_AND_CYCLE_START_ILPB
144   LD      M71  ; MAIN_AUTO_CYCLE_ON
      OUT     M301  ; CYCLE START ILPB
      OUT     M306
; AMBER_TOWER_LAMP_PLC_HEALTHY
163   LD      M70  ; PLC_HEALTHY_MEM_BIT
      OUT     M305
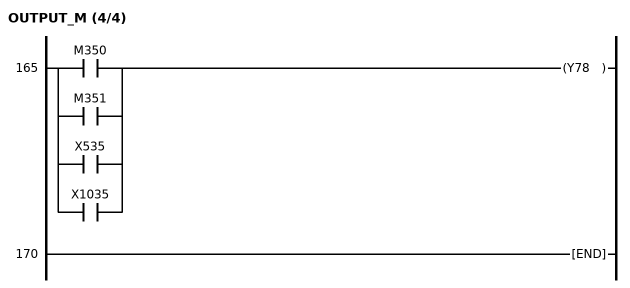
165   LD      M350
      OR      M351
      OR      X535
      OR      X1035
      OUT     Y78
170   END
END_PROGRAM

PROGRAM ROBOT_3
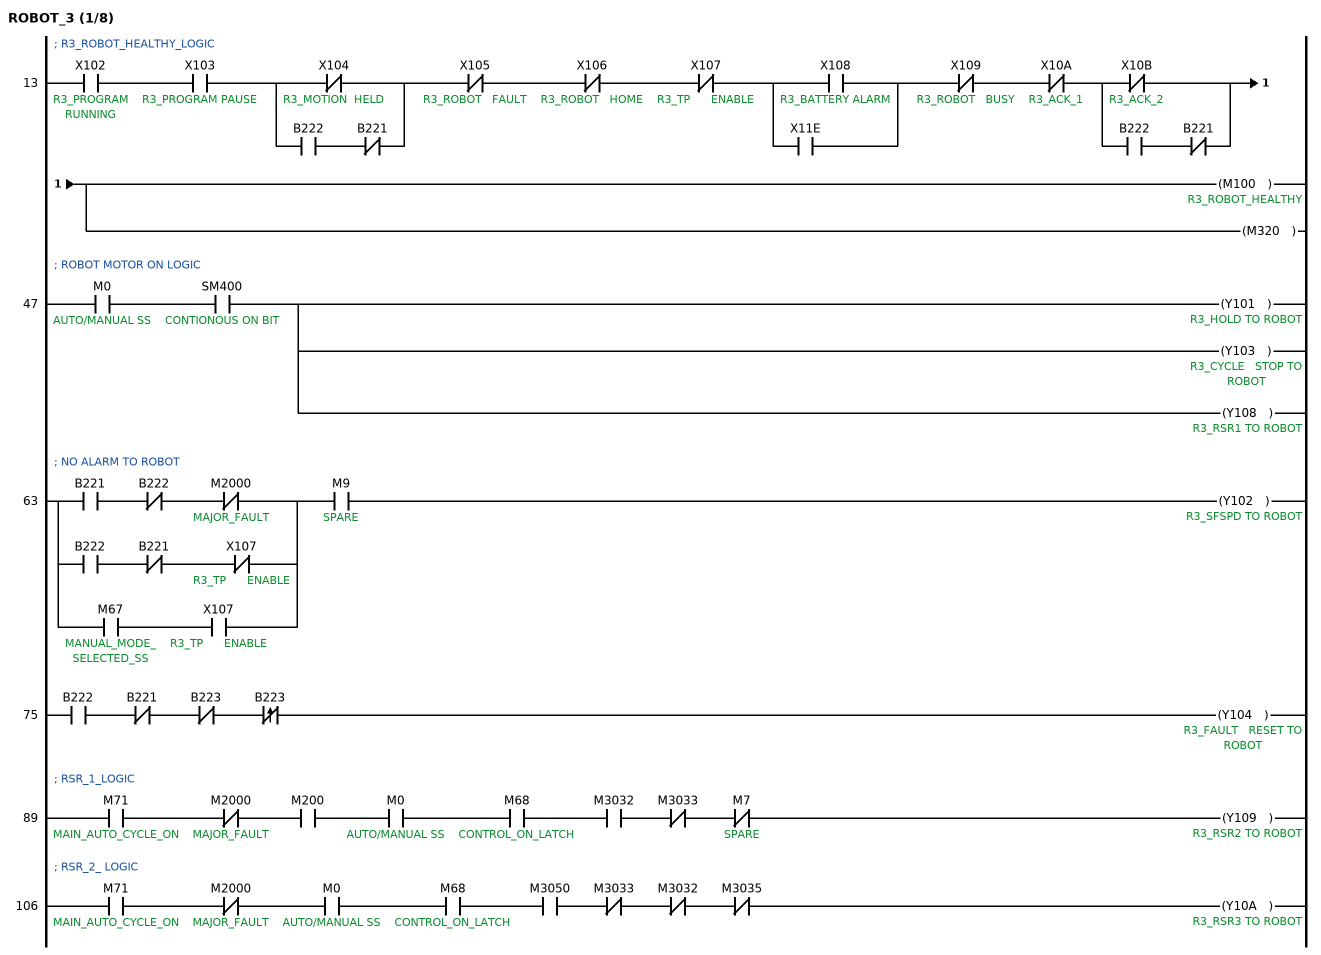
; R3_ROBOT_HEALTHY_LOGIC
13    LD      X102  ; R3_PROGRAM RUNNING
      AND     X103  ; R3_PROGRAM PAUSE
      LDI     X104  ; R3_MOTION  HELD
      LD      B222
      ANI     B221
      ORB
      ANB
      ANI     X105  ; R3_ROBOT   FAULT
      ANI     X106  ; R3_ROBOT   HOME
      ANI     X107  ; R3_TP      ENABLE
      LD      X108  ; R3_BATTERY ALARM
      OR      X11E
      ANB
      ANI     X109  ; R3_ROBOT   BUSY
      ANI     X10A  ; R3_ACK_1
      LDI     X10B  ; R3_ACK_2
      LD      B222
      ANI     B221
      ORB
      ANB
      OUT     M100  ; R3_ROBOT_HEALTHY
      OUT     M320
; ROBOT MOTOR ON LOGIC
47    LD      M0  ; AUTO/MANUAL SS
      AND     SM400  ; CONTIONOUS ON BIT
      OUT     Y101  ; R3_HOLD TO ROBOT
      OUT     Y103  ; R3_CYCLE   STOP TO ROBOT
      OUT     Y108  ; R3_RSR1 TO ROBOT
; NO ALARM TO ROBOT
63    LD      B221
      ANI     B222
      ANI     M2000  ; MAJOR_FAULT
      LD      B222
      ANI     B221
      ANI     X107  ; R3_TP      ENABLE
      ORB
      LD      M67  ; MANUAL_MODE_SELECTED_SS
      AND     X107  ; R3_TP      ENABLE
      ORB
      AND     M9  ; SPARE
      OUT     Y102  ; R3_SFSPD TO ROBOT
75    LD      B222
      ANI     B221
      ANI     B223
      ANDPI   B223
      OUT     Y104  ; R3_FAULT   RESET TO ROBOT
; RSR_1_LOGIC
89    LD      M71  ; MAIN_AUTO_CYCLE_ON
      ANI     M2000  ; MAJOR_FAULT
      AND     M200
      AND     M0  ; AUTO/MANUAL SS
      AND     M68  ; CONTROL_ON_LATCH
      AND     M3032
      ANI     M3033
      ANI     M7  ; SPARE
      OUT     Y109  ; R3_RSR2 TO ROBOT
; RSR_2_ LOGIC
106   LD      M71  ; MAIN_AUTO_CYCLE_ON
      ANI     M2000  ; MAJOR_FAULT
      AND     M0  ; AUTO/MANUAL SS
      AND     M68  ; CONTROL_ON_LATCH
      AND     M3050
      ANI     M3033
      ANI     M3032
      ANI     M3035
      OUT     Y10A  ; R3_RSR3 TO ROBOT
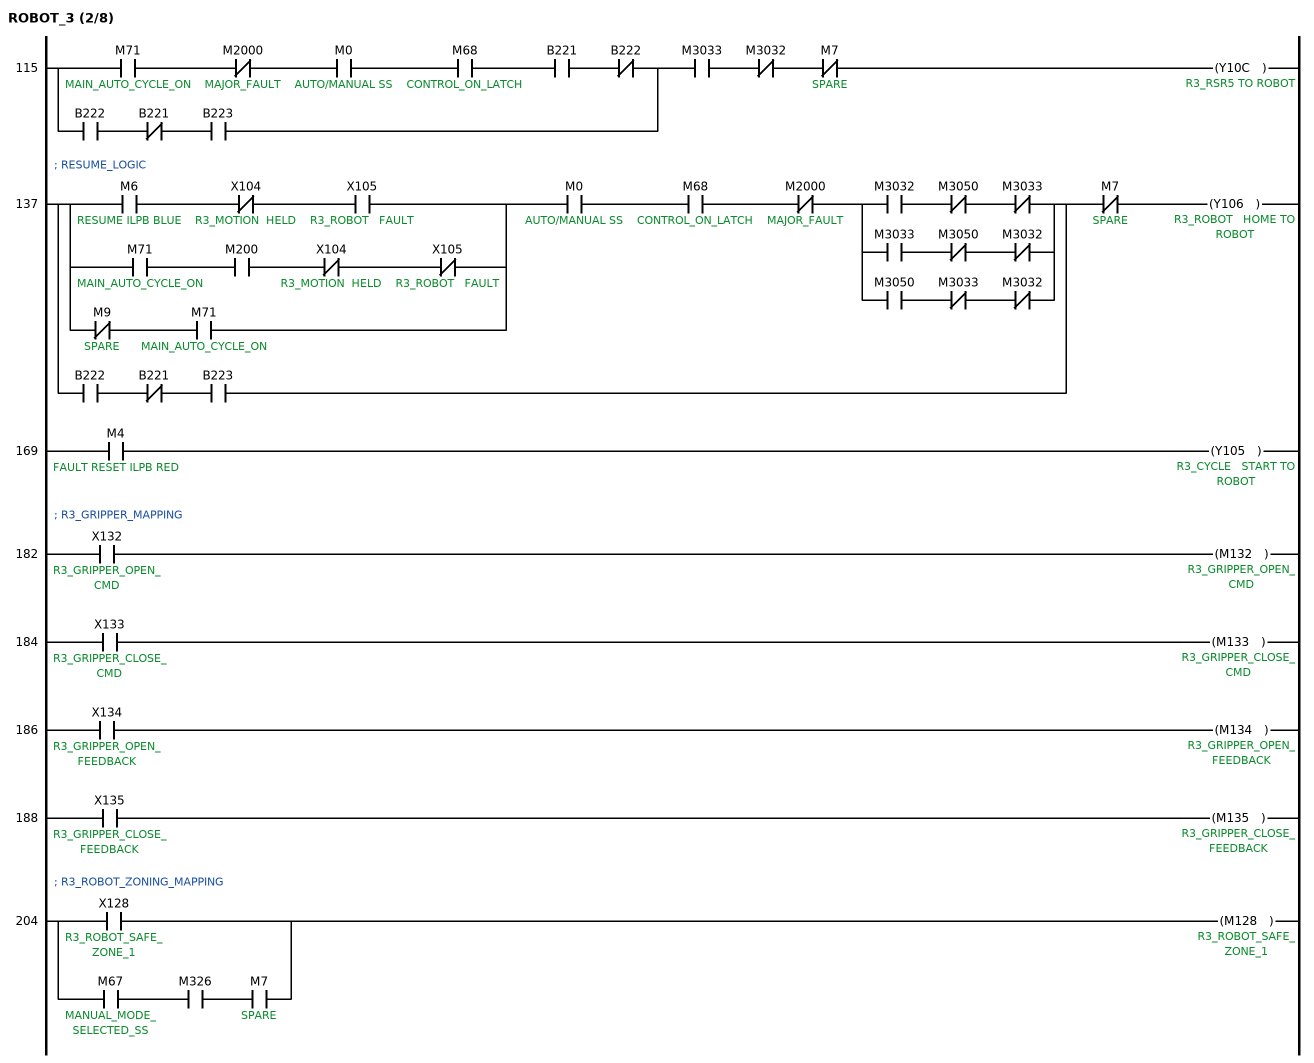
115   LD      M71  ; MAIN_AUTO_CYCLE_ON
      ANI     M2000  ; MAJOR_FAULT
      AND     M0  ; AUTO/MANUAL SS
      AND     M68  ; CONTROL_ON_LATCH
      AND     B221
      ANI     B222
      LD      B222
      ANI     B221
      AND     B223
      ORB
      AND     M3033
      ANI     M3032
      ANI     M7  ; SPARE
      OUT     Y10C  ; R3_RSR5 TO ROBOT
; RESUME_LOGIC
137   LD      M6  ; RESUME ILPB BLUE
      ANI     X104  ; R3_MOTION  HELD
      AND     X105  ; R3_ROBOT   FAULT
      LD      M71  ; MAIN_AUTO_CYCLE_ON
      AND     M200
      ANI     X104  ; R3_MOTION  HELD
      ANI     X105  ; R3_ROBOT   FAULT
      ORB
      LDI     M9  ; SPARE
      AND     M71  ; MAIN_AUTO_CYCLE_ON
      ORB
      AND     M0  ; AUTO/MANUAL SS
      AND     M68  ; CONTROL_ON_LATCH
      ANI     M2000  ; MAJOR_FAULT
      LD      M3032
      ANI     M3050
      ANI     M3033
      LD      M3033
      ANI     M3050
      ANI     M3032
      ORB
      LD      M3050
      ANI     M3033
      ANI     M3032
      ORB
      ANB
      LD      B222
      ANI     B221
      AND     B223
      ORB
      ANI     M7  ; SPARE
      OUT     Y106  ; R3_ROBOT   HOME TO ROBOT
169   LD      M4  ; FAULT RESET ILPB RED
      OUT     Y105  ; R3_CYCLE   START TO ROBOT
; R3_GRIPPER_MAPPING
182   LD      X132  ; R3_GRIPPER_OPEN_CMD
      OUT     M132  ; R3_GRIPPER_OPEN_CMD
184   LD      X133  ; R3_GRIPPER_CLOSE_CMD
      OUT     M133  ; R3_GRIPPER_CLOSE_CMD
186   LD      X134  ; R3_GRIPPER_OPEN_FEEDBACK
      OUT     M134  ; R3_GRIPPER_OPEN_FEEDBACK
188   LD      X135  ; R3_GRIPPER_CLOSE_FEEDBACK
      OUT     M135  ; R3_GRIPPER_CLOSE_FEEDBACK
; R3_ROBOT_ZONING_MAPPING
204   LD      X128  ; R3_ROBOT_SAFE_ZONE_1
      LD      M67  ; MANUAL_MODE_SELECTED_SS
      AND     M326
      AND     M7  ; SPARE
      ORB
      OUT     M128  ; R3_ROBOT_SAFE_ZONE_1
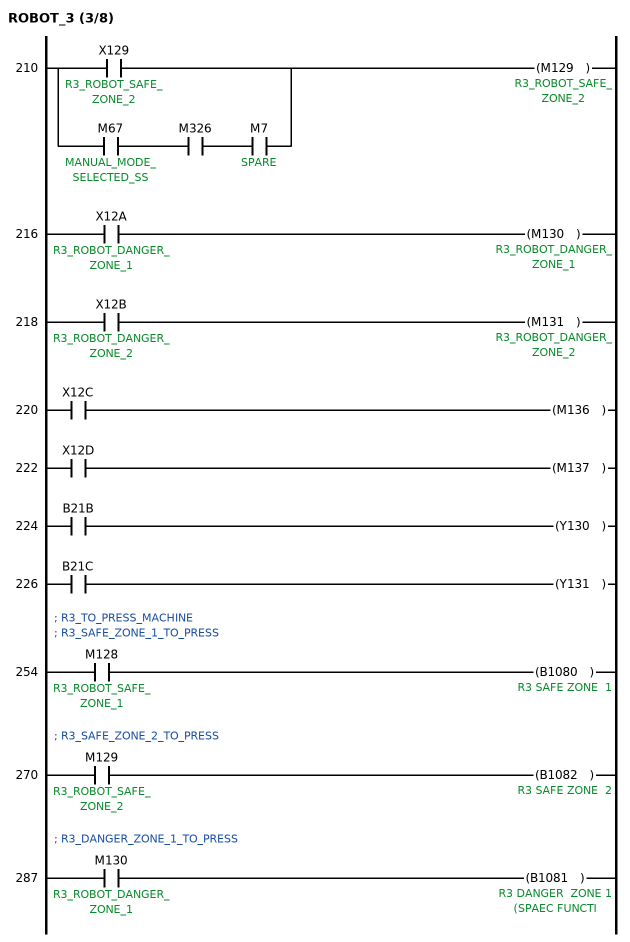
210   LD      X129  ; R3_ROBOT_SAFE_ZONE_2
      LD      M67  ; MANUAL_MODE_SELECTED_SS
      AND     M326
      AND     M7  ; SPARE
      ORB
      OUT     M129  ; R3_ROBOT_SAFE_ZONE_2
216   LD      X12A  ; R3_ROBOT_DANGER_ZONE_1
      OUT     M130  ; R3_ROBOT_DANGER_ZONE_1
218   LD      X12B  ; R3_ROBOT_DANGER_ZONE_2
      OUT     M131  ; R3_ROBOT_DANGER_ZONE_2
220   LD      X12C
      OUT     M136
222   LD      X12D
      OUT     M137
224   LD      B21B
      OUT     Y130
226   LD      B21C
      OUT     Y131
; R3_TO_PRESS_MACHINE
; R3_SAFE_ZONE_1_TO_PRESS
254   LD      M128  ; R3_ROBOT_SAFE_ZONE_1
      OUT     B1080  ; R3 SAFE ZONE  1
; R3_SAFE_ZONE_2_TO_PRESS
270   LD      M129  ; R3_ROBOT_SAFE_ZONE_2
      OUT     B1082  ; R3 SAFE ZONE  2
; R3_DANGER_ZONE_1_TO_PRESS
287   LD      M130  ; R3_ROBOT_DANGER_ZONE_1
      OUT     B1081  ; R3 DANGER  ZONE 1 (SPAEC FUNCTI
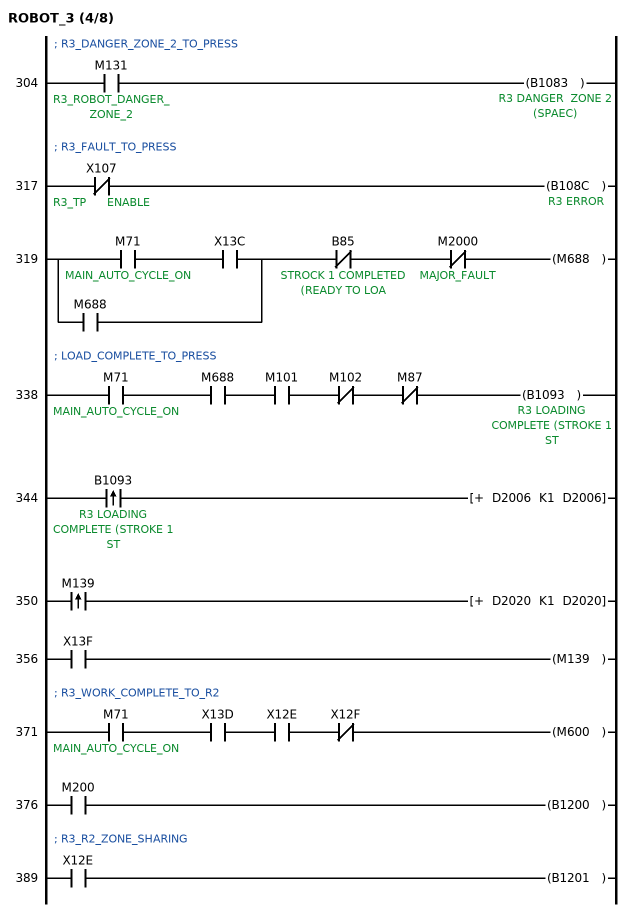
; R3_DANGER_ZONE_2_TO_PRESS
304   LD      M131  ; R3_ROBOT_DANGER_ZONE_2
      OUT     B1083  ; R3 DANGER  ZONE 2 (SPAEC)
; R3_FAULT_TO_PRESS
317   LDI     X107  ; R3_TP      ENABLE
      OUT     B108C  ; R3 ERROR
319   LD      M71  ; MAIN_AUTO_CYCLE_ON
      AND     X13C
      OR      M688
      ANI     B85  ; STROCK 1 COMPLETED (READY TO LOA
      ANI     M2000  ; MAJOR_FAULT
      OUT     M688
; LOAD_COMPLETE_TO_PRESS
338   LD      M71  ; MAIN_AUTO_CYCLE_ON
      AND     M688
      AND     M101
      ANI     M102
      ANI     M87
      OUT     B1093  ; R3 LOADING COMPLETE (STROKE 1 ST
344   LDP     B1093  ; R3 LOADING COMPLETE (STROKE 1 ST
      +       D2006 K1 D2006
350   LDP     M139
      +       D2020 K1 D2020
356   LD      X13F
      OUT     M139
; R3_WORK_COMPLETE_TO_R2
371   LD      M71  ; MAIN_AUTO_CYCLE_ON
      AND     X13D
      AND     X12E
      ANI     X12F
      OUT     M600
376   LD      M200
      OUT     B1200
; R3_R2_ZONE_SHARING
389   LD      X12E
      OUT     B1201
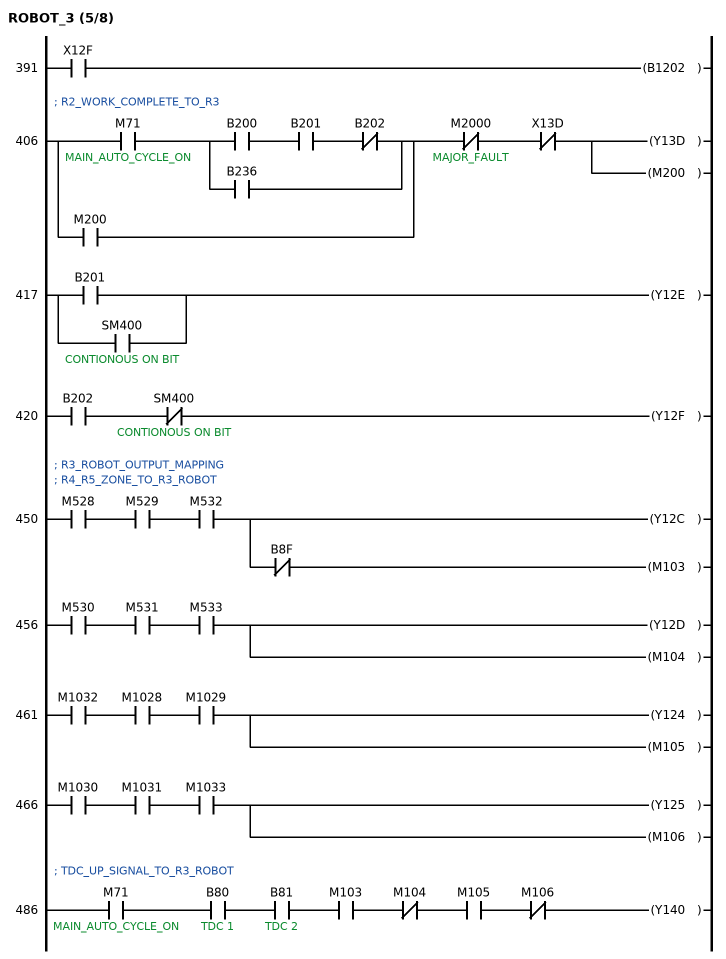
391   LD      X12F
      OUT     B1202
; R2_WORK_COMPLETE_TO_R3
406   LD      M71  ; MAIN_AUTO_CYCLE_ON
      LD      B200
      AND     B201
      ANI     B202
      OR      B236
      ANB
      OR      M200
      ANI     M2000  ; MAJOR_FAULT
      ANI     X13D
      OUT     Y13D
      OUT     M200
417   LD      B201
      OR      SM400  ; CONTIONOUS ON BIT
      OUT     Y12E
420   LD      B202
      ANI     SM400  ; CONTIONOUS ON BIT
      OUT     Y12F
; R3_ROBOT_OUTPUT_MAPPING
; R4_R5_ZONE_TO_R3_ROBOT
450   LD      M528
      AND     M529
      AND     M532
      OUT     Y12C
      ANI     B8F
      OUT     M103
456   LD      M530
      AND     M531
      AND     M533
      OUT     Y12D
      OUT     M104
461   LD      M1032
      AND     M1028
      AND     M1029
      OUT     Y124
      OUT     M105
466   LD      M1030
      AND     M1031
      AND     M1033
      OUT     Y125
      OUT     M106
; TDC_UP_SIGNAL_TO_R3_ROBOT
486   LD      M71  ; MAIN_AUTO_CYCLE_ON
      AND     B80  ; TDC 1
      AND     B81  ; TDC 2
      AND     M103
      ANI     M104
      AND     M105
      ANI     M106
      OUT     Y140
